{attribute 'OPC.UA.DA.StructuredType' := '1'}
FUNCTION_BLOCK FB_OxygenInjector EXTENDS FB_BaseDevice IMPLEMENTS I_Device

VAR
	
	{attribute 'OPC.UA.DA' := '1'} 
	bInContactor AT %I*: BOOL := FALSE;
	{attribute 'OPC.UA.DA' := '1'} 
	bOutContactor AT %Q*: BOOL := FALSE;
	
	{attribute 'OPC.UA.DA' := '0'} 
	eSMState: (WAIT, TURNING_ON, ON, TURNING_OFF, OFF);
	
	{attribute 'OPC.UA.DA' := '0'} 
	tActionTimeout: TIME := T#5S;
	{attribute 'OPC.UA.DA' := '0'} 
	fbTON_timeout: TON := (PT := tActionTimeout, IN := FALSE);
END_VAR

fbTONstartTime();
fbTONstopTime();

IF GVL.bAutoUpdateDeviceState THEN
	eState := eStateTarget;	
END_IF

IF eMode = E_DeviceMode.AUTO AND (eStateTarget = E_DeviceState.ON) THEN
	bEnable := TRUE;
END_IF

IF eMode = E_DeviceMode.MANUAL THEN
	bEnable := TRUE;
END_IF

IF (bEnable AND (eStateTarget = E_DeviceState.ON)) AND eSMState <> ON THEN
		eSMState := TURNING_ON;
END_IF

IF ((bEnable = FALSE) OR (eStateTarget = E_DeviceState.OFF)) AND eSMState <> OFF THEN
		eSMState := TURNING_OFF;
END_IF



CASE eSMState OF
	
	WAIT:
		//Wait for method call to change ESMState
		eState := E_DeviceState.OFF;
		bOutContactor := FALSE;
		
	TURNING_ON: 
		eState := E_DeviceState.TURNING_ON;
		eSMState := ON;
		bOutContactor := TRUE;
	
	ON:
		eState := E_DeviceState.ON;
		bOutContactor := TRUE;
		
		
	TURNING_OFF:

		bOutContactor := FALSE;
		eSMState := OFF;
		
		
	OFF:
		eState := E_DeviceState.OFF;
		bOutContactor := FALSE;
		
END_CASE

{warning 'add method implementation '}
METHOD disable : BOOL
bEnable := FALSE;
END_METHOD

{warning 'add method implementation '}
METHOD enable : BOOL
bEnable := TRUE;
END_METHOD

METHOD FB_init : BOOL
VAR_INPUT
	bInitRetains : BOOL; // if TRUE, the retain variables are initialized (warm start / cold start)
	bInCopyCode : BOOL;  // if TRUE, the instance afterwards gets moved into the copy code (online change)
	
	UnitID: STRING(80);
	UnitDescr: STRING(255); 
END_VAR
sID := UnitID;
sDescr := UnitDescr;
END_METHOD

METHOD setOff : BOOL
VAR_INPUT
END_VAR
eStateTarget := E_DeviceState.OFF;
END_METHOD

METHOD setOn : BOOL
VAR_INPUT
END_VAR
eStateTarget := E_DeviceState.ON;
END_METHOD

END_FUNCTION_BLOCK

(* stored: Version 1.1.0.1, ProductVersion 3.1.4024.12
   POU FB_OxygenInjector: Id {668e5d45-802e-42ce-9ddc-d94c74748a0f}, SpecialFunc None
   Method disable: Id {82040bb5-71ab-4d86-a794-fbb58cb5f5e0}
   Method enable: Id {49a84da0-ad12-43f5-9c2e-92c3330955d7}
   Method FB_init: Id {5f642094-3fe8-470e-b726-75950d4bfae4}
   Method setOff: Id {915557b5-a8ae-40a8-a503-2cceae72eb35}
   Method setOn: Id {5726c980-29e3-4f0e-8f81-7222163776cc} *)
